// TwinCAT 3 PLC project Untitled2
// ProgramVersion: 3.1.4023.0
// libraries:
//   Tc2_Standard, * (Beckhoff Automation GmbH)
//   Tc2_System, * (Beckhoff Automation GmbH)
//   Tc3_Module, * (Beckhoff Automation GmbH)
// project tree:
//   / PlcTask.TcTTO
//   POUs/ FB_Cylinder.TcPOU, FB_DefineAlarm.TcPOU, FB_Test2.TcPOU, FB_Test3.TcPOU, FB_TestFunction.TcPOU, MAIN.TcPOU
// real-time tasks:
//   TASK PlcTask: cycle T#10ms, priority 20, ADS port 350

CONFIGURATION Untitled2
    RESOURCE PLC ON TwinCAT3
        TASK PlcTask(INTERVAL := T#10ms, PRIORITY := 20);
        PROGRAM MAIN WITH PlcTask : MAIN;
    END_RESOURCE
END_CONFIGURATION

// ---- POUs/MAIN.TcPOU
PROGRAM MAIN
VAR
	fbCylinder 		: 	FB_Cylinder;
	fbCylinder1 	: 	FB_Cylinder;
	fbCylinder2 	: 	FB_Cylinder;
	fbTest			:	FB_TestFunction;
	fbTest2			:	FB_Test2;
	fbTest3			:	FB_Test3;
	
	
	Cmd_GoToHP 		: 	BOOL;
	Cmd_GoToWP 		: 	BOOL;
	
END_VAR

fbCylinder();

IF Cmd_GoToHP THEN
	fbCylinder.GoToHP();
	Cmd_GoToHP := FALSE;
ELSIF Cmd_GoToWP THEN
	fbCylinder.GoToWP();
	Cmd_GoToWP := FALSE;	
END_IF

//SafetyIO.Common.Q_Safety_Run[1] := TRUE;
//SafetyIO.Common.Q_Safety_ErrorACK[1] := SafetyIO.I074_Btn_Reset;

(*
fbCylinder(I_IsHP := Pal01_EK.I_613_3V2_HP,
	I_ISWP := Pal01_EK.I_614_3V2_WP,
	I_GoToHP 	:= Cmd_GoToHP,
	I_GoToWP 	:= Cmd_GoToWP,
	Q_CoilToHP => ValveTerminal.YV9_HP,
	Q_CoilToWP => ValveTerminal.YV9_WP
	);
*)

END_PROGRAM

// ---- POUs/FB_Cylinder.TcPOU
FUNCTION_BLOCK FB_Cylinder
VAR_INPUT
	I_GoToHP 	:	BOOL;
	I_GoToWP 	:	BOOL;
	bSensorHP	:	BOOL;
	bSensorWP	:	BOOL;
	
END_VAR
VAR_OUTPUT
	Q_CoilToHP : BOOL;
	Q_CoilToWP : BOOL;
END_VAR
VAR
	bEnable			:	BOOL 	:= TRUE;
	bConfirmError	:	BOOL;

	bSensorWP_check	:	BOOL;
	bSensorHP_check	:	BOOL;
	Cmd_ToHP_act	:	BOOL;
	Cmd_ToWP_act	:	BOOL;

	TON_HP	:	TON;
	TON_WP	:	TON;
	timeHP	:	TIME := T#5S;
	timeWP	:	TIME := T#5S;
	
	iError	:	INT;
	sError	:	STRING;

END_VAR

ConfirmError();

IF bEnable  THEN
	TON_HP(IN := Cmd_ToHP_act, PT := timeHP);
	TON_WP(IN := Cmd_ToWP_act, PT := timeWP);

	CheckErrors();
END_IF

ACTION ConfirmError:
(*
IF SafetyIO.Common.Q_Safety_ErrorACK[1]  THEN
	Enable := TRUE;
END_IF
*)


IF bConfirmError THEN
	bEnable := TRUE;
	iError := 0;
	Cmd_ToHP_act := FALSE;
	Cmd_ToWP_act := FALSE;
	bConfirmError := FALSE;
END_IF
END_ACTION

ACTION GoToHP:
IF bEnable  THEN
	Q_CoilToHP 	:=	TRUE;
	Q_CoilToWP	:= 	FALSE;
	Cmd_ToHP_act:=	TRUE;
END_IF
END_ACTION

ACTION GoToWP:
IF bEnable  THEN
	Q_CoilToHP 	:=	FALSE;
	Q_CoilToWP	:= 	TRUE;
	Cmd_ToWP_act:=	TRUE;
END_IF
END_ACTION

ACTION CheckErrors:
IF bSensorWP THEN
	bSensorWP_check	:= TRUE;
ELSIF bSensorHP THEN
	bSensorHP_check	:= TRUE;
END_IF

//Control Errors for WP
IF TON_WP.Q AND NOT bSensorWP THEN
	IF bSensorWP_check THEN
		iError := 3;
		bSensorWP_check := FALSE;
	ELSE
		iError := 1;
	END_IF
	
//Control Errors for HP
ELSIF TON_HP.Q AND NOT bSensorHP THEN
	IF bSensorHP_check THEN
		iError := 4;
		bSensorHP_check := FALSE;
	ELSE
		iError := 2;
	END_IF
	
//Control for 'Both sensors error'
ELSIF
	bSensorHP AND bSensorWP THEN
	iError := 5;
END_IF

IF iError <> 0 THEN
	bEnable := FALSE;
END_IF

CASE iError OF
	0:	sError := 'OK';
	1:	sError := 'ERROR: Cylinder didnt reach WP on time';
	2:	sError := 'ERROR: Cylinder didnt reach HP on time';
	3:	sError := 'ERROR: Cylinder leaved HP';
	4:	sError := 'ERROR: Cylinder leaved WP';
	5:	sError := 'ERROR: Both sensors for HP and WP activated';
	
END_CASE
END_ACTION

END_FUNCTION_BLOCK

// ---- POUs/FB_TestFunction.TcPOU
FUNCTION_BLOCK FB_TestFunction
VAR_INPUT
	n : int;
END_VAR
VAR_OUTPUT
END_VAR
VAR
END_VAR

n := 0;

END_FUNCTION_BLOCK

// ---- POUs/FB_Test2.TcPOU
FUNCTION_BLOCK FB_Test2
VAR_INPUT
END_VAR
VAR_OUTPUT
END_VAR
VAR
END_VAR

END_FUNCTION_BLOCK

// ---- POUs/FB_Test3.TcPOU
FUNCTION_BLOCK FB_Test3
VAR_INPUT
END_VAR
VAR_OUTPUT
END_VAR
VAR
END_VAR

END_FUNCTION_BLOCK

// ---- POUs/FB_DefineAlarm.TcPOU
FUNCTION_BLOCK FB_DefineAlarm
VAR_INPUT
	
	stEventEntry 		:	TcEventEntry;
	bWithConfirmation 	:	BOOL;
	ipSourceInfo		:	I_TcSourceInfo;
	I_input				:	BOOL;
	
END_VAR
VAR_OUTPUT
END_VAR
VAR
	
	fbTcAlarm			:	FB_TcAlarm;
	I_input_RT			:	R_TRIG;
	ClearAlarm_RT		:	R_TRIG;
	
END_VAR

I_input_RT(CLK := I_input);

IF I_input_RT.Q THEN
	
	fbTcAlarm.createEx(stEventEntry, bWithConfirmation, ipSourceInfo);
	fbTcAlarm.Raise(0);
	
END_IF


IF	Inputs.btn_ClearAlarm THEN
	
	fbTcAlarm.Clear (0, FALSE);
	
END_IF

END_FUNCTION_BLOCK
